Staubli VAL3: Home.dtx

mdesc mNomSpeed
bool bUserRefresh
bool bListRefresh
num nSelected
string sItem
bool bExit
string sParameter
string sListItemValue
string sList
num nType
mdesc mHome = {accel=10, decel=10, tmax=100, leave=1, reach=1, blend=cartesian}
